{attribute 'GeneratedUsingTerminal: AES-D-BC-ECAT-0000'}
{attribute addProperty BoxType "AES-D-BC-ECAT-0000"}
{attribute addProperty Id "InputsInputs_23559BB032OutputsOutputs_FC2FACAD32"}
{attribute addProperty CRC "2239253287"}
{attribute addProperty Size "64"}
TYPE Module_1_32_Byte_Valve_Unit_0x7F_85784B27 :
STRUCT
	{attribute addProperty Name "Inputs"}
	Inputs  : Inputs_23559BB0;
	{attribute addProperty Name "Outputs"}
	Outputs  : Outputs_FC2FACAD;
END_STRUCT
END_TYPE

(* stored: Version 1.2.0.0, ProductVersion 3.1.4024.11
   DUT Module_1_32_Byte_Valve_Unit_0x7F_85784B27: Id {f47022dc-1df6-06cd-3e0a-ee48cacda23d} *)
